(* CoDeSys 2.3 export: PUMP_KD1.EXP *)

(* POU PRG/Pump_KD1, ST *)
PROGRAM Pump_KD1
VAR
	Pump : DRIVE;
END_VAR
;
END_PROGRAM
